FUNCTION_BLOCK MUX_DINT (* See MUX_ANY *)
  (* Standard: 61131-3 *)
  (* Version 0.0, 2004-12-15, JHC, Rockwell Automation, Converted from SRC format. *)
  (* Compiler header: package fb.rt.plc.select; *)
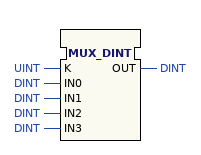
  VAR_INPUT
    K : UINT;
    IN0 : DINT;
    IN1 : DINT;
    IN2 : DINT;
    IN3 : DINT;
  END_VAR
  VAR_OUTPUT
    OUT : DINT;
  END_VAR
END_FUNCTION_BLOCK
